{attribute addProperty BoxType "EPP9022-0060-0017"}
{attribute addProperty Id "StatusAT %I*Status_F11BD7561621VoltageAT %I*DINT32417CurrentAT %I*DINT32418"}
{attribute addProperty CRC "434444532"}
{attribute addProperty SizeInBites "80"}
{attribute addProperty SizeInBytes "10"}
TYPE EPM_Inputs_Channel_19E518F4 :
STRUCT
	{attribute addProperty Name "Status"}
	Status AT %I* : Status_F11BD756;
	{attribute addProperty Name "Voltage"}
	Voltage AT %I* : DINT;
	{attribute addProperty Name "Current"}
	Current AT %I* : DINT;
END_STRUCT
END_TYPE

(* stored: Version 1.2.0.0, ProductVersion 3.1.4024.9
   DUT EPM_Inputs_Channel_19E518F4: Id {a1a0ad29-4b4f-4cd5-94e5-e1be7dc202d7} *)
